// TIA Portal V20 export
TYPE "LER_typeCommunication"
// stored: Access Published
   STRUCT
      ReelCutToStack : "LER_typeCommunicationR2SData";
      StackToReelCut : "LER_typeCommunicationS2RData";
   END_STRUCT;
END_TYPE
